SUBAPPLICATION Uebung_225b (* Dreieck-Sollwertmarker (wie Uebung_225, aber mit dem wiederverwendbaren PositionMarkerFS-Baustein statt F_ADD_Center/F_REAL_TO_INT_Pos/Q_ChildPosition_Dreieck) *)
  (* Standard: 61499-2; Description: Copyright (c) 2026 Meisterschulen am Ostbahnhof This program and the accompanying materials are made available under the terms of the Eclipse Public License 2.0 which is available at https://www.eclipse.org/legal/epl-2.0/ SPDX-License-Identifier: EPL-2.0 *)
  (* Version 1.1, 2026-09-06, Franz Höpfinger, Meisterschulen am Ostbahnhof, Enable xScale on Marker_Dreieck *)
  (* Version 1.0, 2026-09-05, Franz Höpfinger, Meisterschulen am Ostbahnhof, variant of Uebung_225_AX using the reusable PositionMarkerFS block instead of the inline F_ADD/F_REAL_TO_INT/Q_ChildPosition triplet *)
  PACKAGE Uebungen;
  IMPORT Uebungen::const::UT::Dreieck::DefaultPool_Dreieck_PositionMarker::Container_PositionMarker;
  IMPORT Uebungen::const::UT::Dreieck::DefaultPool_Dreieck_Numeric::NumberVariable_Sollwert_N;
  IMPORT Uebungen::const::UT::Dreieck::DefaultPool_Dreieck_Numeric::NumberVariable_Istwert_N;
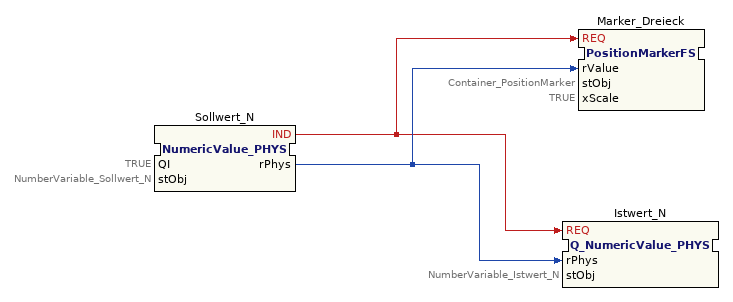
  (* xScale=TRUE auf Marker_Dreieck testet das neue xScale-Flag von Q_ChildPosition (siehe SCALING_FLAG_KONZEPT.md): der Pixel-Offset des Dreieck-Markers wird hier tatsaechlich mit dem DataMask-Scaling-Faktor multipliziert, nicht unveraendert durchgereicht. Diese Uebung (und Uebung_225_AX/227_AX in test_AX) deckt das xScale-Flag also bereits ab - keine reine Doku-Stub-Angelegenheit. *)
  FBS
    Sollwert_N : isobus::UT::io::NumericValue::NumericValue_PHYS(QI := TRUE, stObj := NumberVariable_Sollwert_N);
    Marker_Dreieck : isobus::UT::Q::PositionMarkerFS(stObj := Container_PositionMarker, xScale := TRUE);
    Istwert_N : isobus::UT::Q::Q_NumericValue_PHYS(stObj := NumberVariable_Istwert_N);
  END_FBS
  EVENT_CONNECTIONS
    Sollwert_N.IND TO Marker_Dreieck.REQ;
    Sollwert_N.IND TO Istwert_N.REQ;
  END_CONNECTIONS
  DATA_CONNECTIONS
    Sollwert_N.rPhys TO Marker_Dreieck.rValue;
    Sollwert_N.rPhys TO Istwert_N.rPhys;
  END_CONNECTIONS
END_SUBAPPLICATION
